// TIA Portal V17 export
// export: Created 2023-05-01T07:54:16.8720534Z, ExportSetting WithDefaults, DisplayName Totally Integrated Automation Portal, DisplayVersion V17, DisplayName TIA Portal Openness, DisplayVersion V17, DisplayName TIA Portal Version Control Interface, DisplayVersion V17, DisplayName STEP 7 Professional, DisplayVersion V17, DisplayName STEP 7 Safety, DisplayVersion V17, DisplayName WinCC Advanced / Unified PC, DisplayVersion V17
ORGANIZATION_BLOCK "Main"   // OB1, LAD, ProgramCycle
TITLE = "Main Program Sweep (Cycle)"
{ S7_Optimized_Access := 'TRUE' }
VERSION : 0.1
// stored: AutoNumber true, IsIECCheckEnabled false, SetENOAutomatically false
   VAR_INPUT
      Initial_Call : Bool;   // Initial call of this OB
      Remanence : Bool;   // =True, if remanent data are available
   END_VAR
   VAR_TEMP
      temperature : Real;
   END_VAR
   VAR CONSTANT
      temperatureMin : Real := 0.0;
      temperatureMax : Real := 100.0;
   END_VAR
BEGIN

REGION Network 1: Scale analog input temperature on IW64
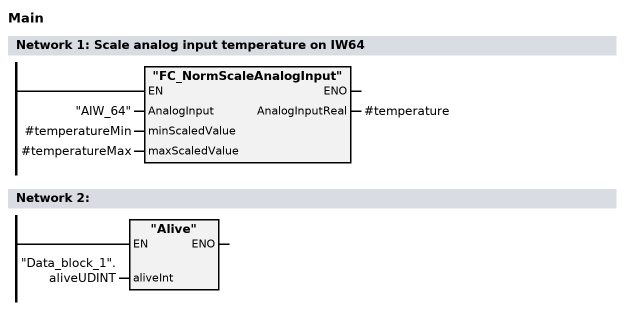
   RUNG wire#powerrail
      "FC_NormScaleAnalogInput"(AnalogInput := "AIW_64", minScaledValue := #temperatureMin, maxScaledValue := #temperatureMax, AnalogInputReal => #temperature)
   END_RUNG
   // the same network as SCL:
   "FC_NormScaleAnalogInput"(AnalogInput := "AIW_64",
                           minScaledValue := #temperatureMin,
                           maxScaledValue := #temperatureMax,
                           AnalogInputReal => #temperature);
END_REGION

REGION Network 2
   RUNG wire#powerrail
      "Alive"(aliveInt := "Data_block_1".aliveUDINT)
   END_RUNG
   // the same network as SCL:
   "Alive"(aliveInt := "Data_block_1".aliveUDINT);
END_REGION
END_ORGANIZATION_BLOCK
